// SIMATIC S7-200 SMART project (STEP 7-Micro/WIN SMART), CPU ST40

SYMBOL_TABLE Table 1
delay            50
END_SYMBOL_TABLE

SYMBOL_TABLE System Symbols
Always_On        SM0.0    // Always ON
First_Scan_On    SM0.1    // ON for the first scan cycle only
END_SYMBOL_TABLE

ORGANIZATION_BLOCK MAIN:OB1
TITLE=Program Comments
BEGIN
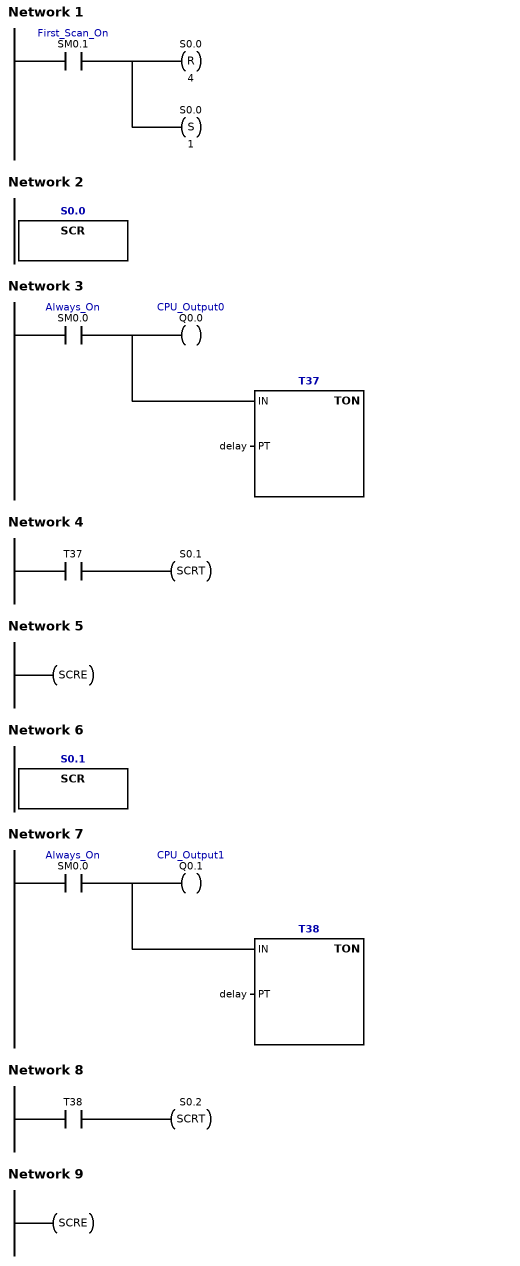
Network 1
LD     First_Scan_On:SM0.1
R      S0.0, 4
S      S0.0, 1
Network 2
LSCR   S0.0
Network 3
LD     Always_On:SM0.0
=      CPU_Output0:Q0.0
TON    T37, delay
Network 4
LD     T37
SCRT   S0.1
Network 5
SCRE
Network 6
LSCR   S0.1
Network 7
LD     Always_On:SM0.0
=      CPU_Output1:Q0.1
TON    T38, delay
Network 8
LD     T38
SCRT   S0.2
Network 9
SCRE
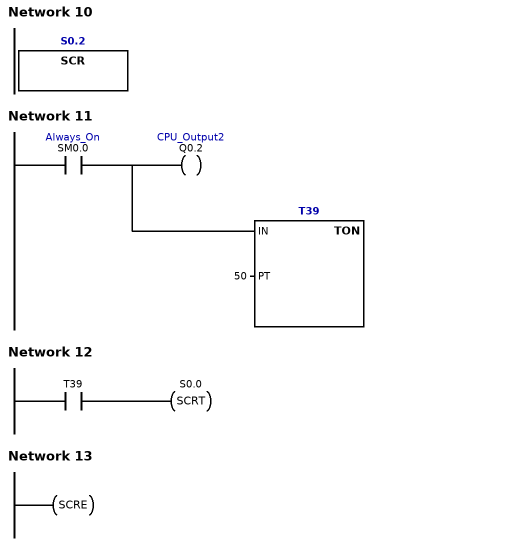
Network 10
LSCR   S0.2
Network 11
LD     Always_On:SM0.0
=      CPU_Output2:Q0.2
TON    T39, 50
Network 12
LD     T39
SCRT   S0.0
Network 13
SCRE
END_ORGANIZATION_BLOCK
